// TIA Portal V17 export
// export: Created 2023-12-22T15:03:19.1586487Z, ExportSetting WithDefaults, DisplayName Totally Integrated Automation Portal, DisplayVersion V17, DisplayName TIA Portal Openness, DisplayVersion V17, DisplayName TIA Portal Version Control Interface, DisplayVersion V17, DisplayName STEP 7 Professional, DisplayVersion V17, DisplayName STEP 7 Safety, DisplayVersion V17, DisplayName WinCC Advanced, DisplayVersion V17
DATA_BLOCK "Any_DB"   // DB11
{ S7_Optimized_Access := 'FALSE' }
VERSION : 0.1
// stored: AutoNumber true, DBAccessibleFromOPCUA true, DBAccessibleFromWebserver true, IsOnlyStoredInLoadMemory false, IsWriteProtectedInAS false
   VAR RETAIN
      SKV_FE_All : Real;
      D { S7_SetPoint := 'True'} : Real := 1.0;
      C { S7_SetPoint := 'True'} : Real := 7.0;
      SP_ELZ : Real;
      SP_1 : Real;
      SP_2 : Real;
   END_VAR
BEGIN
END_DATA_BLOCK
